(* PLC project KinIn_v3.project, CODESYS CODESYS V3.5 SP19 *)
(* stored: creationDateTime 2025-01-20T16:27:59.8633225, modificationDateTime 2025-01-20T16:17:39.6822999 *)

FUNCTION_BLOCK Vect_byScalar
  VAR_INPUT
    {attribute 'variable_length_array_original_scope' := 'Inout'}
    {attribute 'variable_length_array' := 'ARRAY[*] OF REAL'}
    {attribute 'Dimensions' := '1'}
    Vector : POINTER TO REAL;
  END_VAR
  VAR_IN_OUT
    scalar : REAL;
  END_VAR
  VAR_INPUT
    {attribute 'variable_length_array_original_scope' := 'Inout'}
    {attribute 'variable_length_array' := 'ARRAY[*] OF REAL'}
    {attribute 'Dimensions' := '1'}
    VectorByScalar : POINTER TO REAL;
  END_VAR
  VAR
    i : DINT;
  END_VAR

            FOR i:=1 TO UPPER_BOUND(Vector,1) DO
	VectorByScalar[i]:=Vector[i]*scalar;

END_FOR
          
END_FUNCTION_BLOCK
